(* PLC project TestUml.project, Rexroth ctrlX PLC Engineering ctrlX PLC 1.20.12 *)
(* stored: creationDateTime 2025-03-04T16:25:50.9610727, modificationDateTime 2025-03-04T16:13:03.9525114 *)

{attribute 'qualified_only'}
{attribute 'strict'}
TYPE E_Operation : (Idle := 999, AddUp := 10, Substract := 20, Multiply := 30, Divide := 40, Done := 50, Error := 666) UINT;
END_TYPE

TYPE ST_TestAlgo : STRUCT
  Enable : BOOL;
  FirstValue : DINT;
  SecondeValue : DINT;
  Add_1_2 : BOOL;  (* Operation *)
  Sub_1_2 : BOOL;
  Mul_1_2 : BOOL;
  Div_1_2 : BOOL;
END_STRUCT;
END_TYPE

FUNCTION_BLOCK FB_BaseAlgo
  VAR_INPUT
    Enable : BOOL;
    FirstValue : DINT;
    SecondeValue : DINT;
    Add_1_2 : BOOL;  (* Operation *)
    Sub_1_2 : BOOL;
    Mul_1_2 : BOOL;
    Div_1_2 : BOOL;
  END_VAR
  VAR_OUTPUT
    Result : DINT;
    Error : BOOL;
    Done : BOOL;
  END_VAR
  VAR
    eSelectOp : E_Operation;
    testZero : BOOL;
  END_VAR

            IF Enable THEN
	IF Add_1_2 THEN
		eSelectOp := E_Operation.AddUp;
	ELSIF Sub_1_2 THEN
		eSelectOp := E_Operation.Substract;
	ELSIF Mul_1_2 THEN
		eSelectOp := E_Operation.Multiply;
	ELSIF Div_1_2 THEN
		eSelectOp := E_Operation.Divide;
	END_IF
ELSE
	eSelectOp := E_Operation.Idle;
END_IF

CASE eSelectOp OF
	E_Operation.Idle 		:
		;
	E_Operation.AddUp	 	:
		Result := FirstValue + SecondeValue;
	E_Operation.Substract	:
		Result := FirstValue - SecondeValue; 
	E_Operation.Multiply	:
		Result := FirstValue * SecondeValue; 
	E_Operation.Divide		:
		IF SecondeValue = 0 THEN
			eSelectOp := E_Operation.Error;
		ELSE
			Result := FirstValue / SecondeValue; 			
		END_IF
	E_Operation.Done        :
		;
	E_Operation.Error		:
		;
END_CASE
          
END_FUNCTION_BLOCK

PROGRAM PRG_Operation
  VAR
    uliLoop : ULINT;
    fbBaseAlgo : FB_BaseAlgo;
    fbBaseExtended : FB_BaseAlgoExtended;
    stTestAlgo : ST_TestAlgo;
    diResultBase : DINT;
    diResultExtend : DINT;
    fbUseFB_Base_1 : FB_UseFB_Base;  (* Using FB_BaseAlgo *)
    fbUseFB_Base_2 : FB_UseFB_Base;
  END_VAR

            uliLoop := uliLoop + 1;

// Set Base Inputs
fbBaseAlgo.Enable := stTestAlgo.Enable;
fbBaseAlgo.FirstValue := stTestAlgo.FirstValue;
fbBaseAlgo.SecondeValue := stTestAlgo.SecondeValue;

fbBaseAlgo.Add_1_2 := stTestAlgo.Add_1_2;
fbBaseAlgo.Sub_1_2 := stTestAlgo.Sub_1_2;
fbBaseAlgo.Mul_1_2 := stTestAlgo.Mul_1_2;
fbBaseAlgo.Div_1_2 := stTestAlgo.Div_1_2;

// Extended Algo
fbBaseAlgo();
diResultBase := fbBaseAlgo.Result;

// Set Base Inputs
fbBaseExtended.Enable := stTestAlgo.Enable;
fbBaseExtended.FirstValue := stTestAlgo.FirstValue;
fbBaseExtended.SecondeValue := stTestAlgo.SecondeValue;

fbBaseExtended.Add_1_2 := stTestAlgo.Add_1_2;
fbBaseExtended.Sub_1_2 := stTestAlgo.Sub_1_2;
fbBaseExtended.Mul_1_2 := stTestAlgo.Mul_1_2;
fbBaseExtended.Div_1_2 := stTestAlgo.Div_1_2;

// Call base Algo
fbBaseExtended();
diResultExtend := fbBaseExtended.Result;

fbUseFB_Base_1(fb := fbBaseAlgo);
fbUseFB_Base_2(fb := fbBaseExtended);
// End of code
          
END_PROGRAM

FUNCTION_BLOCK FB_BaseAlgoExtended EXTENDS FB_BaseAlgo
  VAR_INPUT
    Square : BOOL;
  END_VAR

            SUPER^();

// What to do with Square ?
// On option is to rewrite the core of FB_BaseAlgo...
          
END_FUNCTION_BLOCK

FUNCTION_BLOCK FB_UseFB_Base
  VAR_IN_OUT
    fb : FB_BaseAlgo;
  END_VAR
  VAR
    iMyLoop : INT;
    diMyResult : DINT;
  END_VAR

            iMyLoop := iMyLoop + 1;

fb();
diMyResult := fb.Result;
          
END_FUNCTION_BLOCK
